Omron CX-Programmer project NewProject (CX-Programmer 9.73)

# PLC NewPLC1: CP1E E20

## Global symbols (name address type ; comment)
0.00 BOOL  ; NO1
0.01 BOOL  ; NO2
0.02 BOOL  ; NO2
0.03 BOOL  ; NO3
0.04 BOOL  ; NO2
0.08 BOOL  ; NO3
1.00 BOOL  ; DORONG
1.01 BOOL  ; NO2
2.00 BOOL  ; TARIK
3.00 BOOL  ; NC2

## Program NewProgram1 (cyclic task 0)

### Section Section1

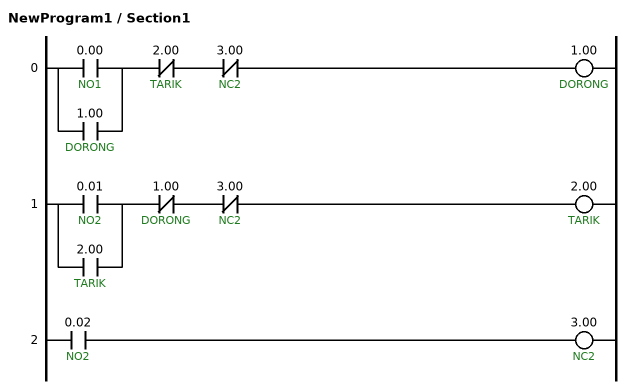
; rung 0
LD 0.00  ; NO1
OR 1.00  ; DORONG
ANDNOT 2.00  ; TARIK
ANDNOT 3.00  ; NC2
OUT 1.00  ; DORONG
; rung 1
LD 0.01  ; NO2
OR 2.00  ; TARIK
ANDNOT 1.00  ; DORONG
ANDNOT 3.00  ; NC2
OUT 2.00  ; TARIK
; rung 2
LD 0.02  ; NO2
OUT 3.00  ; NC2

### Section END
; rung 0
END(001)